# EPICS IOC start-up script: iocsh/ethercatmc2slit.iocsh
dbLoadRecords("ethercatmcslit_soft.template", "P=$(P), SLIT=$(SLIT), mXp=$(mXp), mXn=$(mXn) ")
